Staubli VAL3: getResolution.pgx

public program getResolution(num& x_nResolution[])
begin
  // This routine returns the encoder resolution
  //
  // Input Param
  //
  // Output Param
  //  x_nEncResolution  : Encoder resolution. -1 is returned if not applicable
  //
  //
  //----------------------------------------------------------------
  //
  if ioStatus(aoEncResolution)>=0
    nEncResolution=aioGet(aoEncResolution)
    x_nResolution=nEncResolution
  else
    x_nResolution=-1
  endIf
end
